FUNCTION_BLOCK Test_AssertEquals_INT EXTENDS T_UnitTestBase
VAR
    AssertionUnderTest : T_Assertion;
    INT_Variable : INT := 1111;
END_VAR

// Test the assertion...
AssertionUnderTest.AssertEquals_INT(
    Expected := 2222,
    Actual   := INT_Variable,
    VariableName := 'INT_Variable');
 
// Assert that the assertion failed...
Assertion.AssertEquals_BOOL(Expected     := TRUE,
                            Actual       := AssertionUnderTest.AssertionFailed,
                            VariableName := 'AssertionUnderTest.AssertionFailed');

// Check the assertion worked...  
CheckAssertion(NextState := 0);

END_FUNCTION_BLOCK

(* stored: Version 1.1.0.1, ProductVersion 3.1.4024.11
   POU Test_AssertEquals_INT: Id {20c7f3ec-cc54-4bde-b7dd-b58ce6b65415}, SpecialFunc None *)
